# B&R Automation Studio project ProjetoPadrao2022
Automation Studio 4.1.14.40 SP

## Configuration Config1

CPU X20CP1583, AutomationRuntime G4.09, Build 4.1.2, Vc V4.15.9

### Task classes (Cpu.sw)
```
Cyclic#4 (cycle 100000 us, tolerance 100000 us):
  ProjetoA11 <- ProjetoA110.prg
Libraries: LoopConR, sys_lib, brsystem, Runtime, standard, MTSystem, MTTypes, MTBasics
```

### Hardware
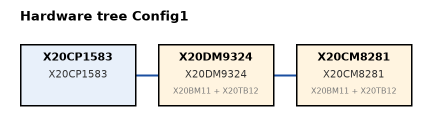
```
X20BM11 : X20BM11 v1.0.0.0  [X2X1 -> X20CP1583.IF6]
X20BM11a : X20BM11 v1.0.0.0  [X2X1 -> X20BM11.X2X2]
X20CM8281 : X20CM8281 v1.0.3.0  [SS1 -> X20TB12a.SS; SL -> X20BM11a.SL1]
X20CP1583 : X20CP1583 v1.0.4.0
  Connector IF2:
    ActivateDevice = 1
    EthInterfaceRedundant = 0
    Mode = Manual
    InternetAddress = 192.168.0.70
    SubnetMask = 255.255.255.0
  Connector IF3:
    EplInterfaceRedundant = 0
    EplEthInterfaceRedundant = 0
  ConfigurationID = ProjetoPadrao2022_Config1
  TimerDeviceType = SWIOTIMER
  Cyclic1Duration = 10000
  Cyclic1Tolerance = 10000
  Cyclic2Duration = 20000
  Cyclic2Tolerance = 20000
  Cyclic3Duration = 50000
  Cyclic3Tolerance = 50000
  Cyclic4Duration = 100000
  Cyclic4Tolerance = 100000
  Cyclic5Duration = 200000
  Cyclic5Tolerance = 200000
  Cyclic6Duration = 500000
  Cyclic6Tolerance = 500000
  Cyclic7Duration = 1000000
  Cyclic7Tolerance = 1000000
  Cyclic8Duration = 10000
  Cyclic8Tolerance = 30000000
  ActivateOpcUa = 1
X20DM9324 : X20DM9324 v1.0.1.0  [SS1 -> X20TB12.SS; SL -> X20BM11.SL1]
X20TB12 : X20TB12 v1.0.0.0
X20TB12a : X20TB12 v1.0.0.0
```

### IoMap.iom - X20CP1583/IoMap.iom
```iecst
(********************************************************************
 * COPYRIGHT --
 ********************************************************************
 * File: IoMap.iom
 * Author: supervisorio
 * Created: September 13, 2022
 ********************************************************************
 * IO mapping file
 ********************************************************************)
VAR_CONFIG
	::ProjetoA11:X AT %IW."X20CM8281".AnalogInput01;
	::ProjetoA11:SAIDA AT %QX."X20DM9324".DigitalOutput01;
	::ProjetoA11:BOTAO_VERMELHO AT %IX."X20DM9324".DigitalInput02;
END_VAR
```

## Logical view

Binary libraries used (declarations not repeated): operator, runtime, astime, AsIecCon, LoopConR 4.10.0, sys_lib, brsystem, standard, MTSystem 1.00.1, MTTypes 1.03.4, MTBasics 2.30.2

### Global.var - Global variables
```iecst
VAR
	LIGA : BOOL;
	ESTADO : INT;
	TEMPERATURA : REAL;
	SETPOINT : REAL;
	KP : REAL;
	TI : REAL;
	TD : REAL;
	SAIDA_PID : REAL;
	MAX_TEMP_PERMITIDA : REAL;
END_VAR
```


### Program Logical/ProjetoA110 (IEC) - Program

#### ProjetoA110Init.st - Initialization code
```iecst
(********************************************************************
 * COPYRIGHT --
 ********************************************************************
 * Program: ProjetoA110
 * File: ProjetoA110Init.st
 * Author: supervisorio
 * Created: November 18, 2023
 ********************************************************************
 * Implementation of program ProjetoA110
 ********************************************************************)

PROGRAM _INIT

	SETPOINT := 50.0;
	MAX_TEMP_PERMITIDA := 75.0;

END_PROGRAM
```

#### ProjetoA110.var - Local variables
```iecst
(********************************************************************
 * COPYRIGHT --
 ********************************************************************
 * Program: ProjetoA110
 * File: ProjetoA110.var
 * Author: supervisorio
 * Created: November 18, 2023
 ********************************************************************
 * Local variables of program ProjetoA110
 ********************************************************************)
VAR
	BOTAO_VERDE : BOOL;
	BOTAO_VERMELHO : BOOL;
	BLOCO_PID : LCRSlimPID;
	X : INT;
	BLOCO_PWM : LCRPWM;
	SAIDA : BOOL;
	PARAMETROS : lcrslimpid_par_typ;
	HABILITA_TRACE : BOOL;
END_VAR
```

#### ProjetoA110Cyclic.st - Cyclic code
```iecst
(********************************************************************
 * COPYRIGHT --
 ********************************************************************
 * Program: ProjetoA110
 * File: ProjetoA110Cyclic.st
 * Author: supervisorio
 * Created: November 18, 2023
 ********************************************************************
 * Implementation of program ProjetoA110
 ********************************************************************)

PROGRAM _CYCLIC
	TEMPERATURA := X / 327.67;

	PARAMETROS.Y_max := 100;
	PARAMETROS.Y_min := 0;

	IF LIGA = TRUE THEN
		BLOCO_PID.enable := TRUE;
		BLOCO_PWM.enable := TRUE;
		HABILITA_TRACE := TRUE;
	END_IF;

	IF EDGENEG(BOTAO_VERMELHO) OR LIGA = FALSE THEN
		BLOCO_PID.enable := FALSE;
		BLOCO_PWM.enable := FALSE;
		HABILITA_TRACE := FALSE;
		LIGA := FALSE;
	END_IF;

	IF ESTADO = 1 THEN
		BLOCO_PID.request := 1;
		KP := 0;
		TI := 0;
		TD := 0;

		IF BLOCO_PID.PIDTune_inst.state = 50 THEN
			ESTADO := 4;
			LIGA := FALSE;
		END_IF;
	ELSIF ESTADO = 3 THEN
		BLOCO_PID.request := 3;
		PARAMETROS.Kp := KP;
		PARAMETROS.Tn := TI;
		PARAMETROS.Tv := TD;
	ELSIF ESTADO = 4 THEN
		BLOCO_PID.request := 4;
		KP := PARAMETROS.Kp;
		TI := PARAMETROS.Tn;
		TD := PARAMETROS.Tv;
	END_IF;

	BLOCO_PID.pPar := ADR(PARAMETROS);
	BLOCO_PID.request := ESTADO;
	BLOCO_PID.W := SETPOINT;
	BLOCO_PID.X := TEMPERATURA;
	BLOCO_PID();

	BLOCO_PWM.max_value := 100;
	BLOCO_PWM.min_value := 0;
	BLOCO_PWM.t_min_pulse := 0;
	BLOCO_PWM.t_period := 1;
	BLOCO_PWM.x := BLOCO_PID.Y;
	BLOCO_PWM();

	SAIDA := BLOCO_PWM.pulse;
	SAIDA_PID := BLOCO_PID.Y;
END_PROGRAM
```
